{attribute 'no_explicit_call' := 'do not call this POU directly'}
{attribute 'conditionalshow_all_locals'}
// Function Block to invoke RPC calls.
FUNCTION_BLOCK FINAL FB_RPC_Dynamic EXTENDS FB_RpcBase IMPLEMENTS I_RpcDynamicConfig

VAR
	{attribute 'hide'}	
	fbConfig				: FB_RpcConfig;
END_VAR

METHOD INTERNAL ConfigDoneCallback : HRESULT
VAR_INPUT CONSTANT
	sAmsNetId		: REFERENCE TO T_AmsNetId;
	nAmsPort		: T_AmsPort;
	sInstancePath	: REFERENCE TO STRING;
	sSymbol			: REFERENCE TO STRING;
END_VAR
VAR
	sRpcSymbol : T_MaxString;
END_VAR
IF sAmsNetId = '' THEN
	ConfigDoneCallback := E_HRESULTAdsErr.INVALIDPARM;
	RETURN;
END_IF

IF nAmsPort = 0 THEN
	ConfigDoneCallback := E_HRESULTAdsErr.INVALIDPARM;
	RETURN;
END_IF

IF sInstancePath = '' THEN
	ConfigDoneCallback := E_HRESULTAdsErr.INVALIDPARM;
	RETURN;
END_IF

IF sSymbol = '' THEN
	ConfigDoneCallback := E_HRESULTAdsErr.INVALIDPARM;
	RETURN;
END_IF

IF sAmsNetId <> SUPER^.sAmsNetId THEN
	SUPER^.ReleaseHandle();
	SUPER^.sAmsNetId := sAmsNetId;	
END_IF

IF nAmsPort <> SUPER^.nAmsPort THEN
	SUPER^.ReleaseHandle();
	SUPER^.nAmsPort := nAmsPort;	
END_IF

sRpcSymbol := F_RpcSymbol(sInstancePath:= sInstancePath, sSymbolName:= sSymbol);
IF sRpcSymbol <> SUPER^.sRpcSymbolField THEN
	SUPER^.ReleaseHandle();
	SUPER^.sRpcSymbol := sRpcSymbol;
END_IF;

ConfigDoneCallback := S_OK;
END_METHOD

METHOD Configure : I_RpcDynamicConfigAmsNetId
fbConfig.SetCallback(pFbRpcBase:= THIS);
Configure := fbConfig;
END_METHOD

METHOD FB_exit : BOOL
VAR_INPUT
	bInCopyCode : BOOL; // if TRUE, the exit method is called for exiting an instance that is copied afterwards (online change).
END_VAR
IF SUPER^.nSymbolHandle > cNoSymbolNameHandle THEN
	SUPER^.ReleaseHandle();
END_IF
END_METHOD

END_FUNCTION_BLOCK

(* stored: Version 1.1.0.1, ProductVersion 3.1.4024.12
   POU FB_RPC_Dynamic: Id {8d147792-0928-41d9-a8ad-6feec4d91f92}, SpecialFunc None
   Folder ITFs: Id {69f227c9-1e01-43cd-84f0-b192164f0d10}
   Method ConfigDoneCallBack: Id {fbb623cb-6666-478b-ad57-726ac340c777}
   Method Configure: Id {c9c670fa-9394-4404-a82d-1b6ab703eecb}
   Method FB_exit: Id {3877c5a4-13ea-4a21-9447-b91548b15388} *)
